FUNCTION_BLOCK CLIENT_3_0 (* Connect to a SERVER_3 Block *)
  (* Standard: 61499-2; Description: Copyright (c) 2017, 2025 fortiss GmbH , Johannes Kepler University Linz This program and the accompanying materials are made available under the terms of the Eclipse Public License 2.0 which is available at https://www.eclipse.org/legal/epl-2.0/ SPDX-License-Identifier: EPL-2.0 *)
  (* Version 3.0, 2025-19-26, Alois Zoitl, Created from CLIENT_1 *)
  PACKAGE iec61499::net;
  {SET_ATTRIBUTE(eclipse4diac::core::GenericClassName, 'GEN_CLIENT')}
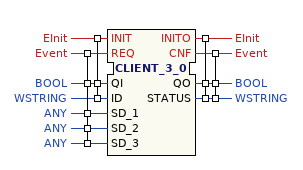
  EVENT_INPUT
    INIT : EInit WITH QI, ID; (* Open new connection (QI = TRUE) / Close connection (QI = FALSE) *)
    REQ WITH QI, SD_1, SD_2, SD_3; (* Send data to Server, Request Data from Server *)
  END_EVENT
  EVENT_OUTPUT
    INITO : EInit WITH QO, STATUS; (* New connection established (QI = TRUE) / connection closed (QI = FALSE) *)
    CNF WITH QO, STATUS; (* New data available from Server *)
  END_EVENT
  VAR_INPUT
    QI : BOOL;
    ID : WSTRING;
    SD_1 : ANY;
    SD_2 : ANY;
    SD_3 : ANY;
  END_VAR
  VAR_OUTPUT
    QO : BOOL;
    STATUS : WSTRING;
  END_VAR
END_FUNCTION_BLOCK
